{attribute 'GeneratedUsingTerminal: EL2521--0000'}
{attribute addProperty BoxType "EL2521--0000"}
{attribute addProperty Id "EtcSlaveTerminalBaseInputsAT %I*Inputs_A33354244OutputsAT %Q*Outputs_8F8B60FA4WcStateAT %I*WcState_9091E0EB2InfoDataAT %I*InfoData_32EB74EA10"}
{attribute addProperty CRC "1692347064"}
{attribute addProperty Size "20"}
TYPE EL2521_64DF2AB8 EXTENDS EtcSlaveTerminalBase :
STRUCT
	{attribute addProperty Name "Inputs"}
	Inputs : Inputs_A3335424;
	{attribute addProperty Name "Outputs"}
	Outputs : Outputs_8F8B60FA;
	{attribute addProperty Name "WcState"}
	WcState : WcState_9091E0EB;
	{attribute addProperty Name "InfoData"}
	InfoData : InfoData_32EB74EA;
END_STRUCT
END_TYPE

(* stored: Version 1.2.0.0, ProductVersion 3.1.4024.9
   DUT EL2521_64DF2AB8: Id {e74cc213-958b-47ff-8f2d-0a0b6a408564} *)
